(*
SPDX-FileCopyrightText: © 2026 Oleksandr Tiutyk <trofimich@gmail.com>
SPDX-License-Identifier: MIT
License: https://opensource.org/license/mit
*)

(*!
<summary>Formats diagnostics for text-file logging and advances file operations through cyclic execution.</summary>
<description>
Use this backend for buffered text-file output. Direct TryLog and Execute calls on one instance must belong to
one task: its message queue, buffers and file-operation state are not synchronized for concurrent access. For
callers in multiple tasks, use QueuedLogger and let its owner task service this backend; do not bypass the
wrapper with concurrent direct calls. Separate instances writing independently must use separate output files.
Cyclic Execute is required to advance writing and cleanup. Exception logging accepts IReadOnlyException and
reads borrowed diagnostics without transferring ownership. Implementations must not retain exception
references beyond their task cleanup. FAILED is terminal for this instance: no automatic retry or recovery is
provided. Continue calling Execute after failure to discard queued messages, cancel active tasks and release
the send buffer once file operations have finished. Pending messages are not retried. The instance must remain
alive during cleanup. Busy reports pending initialization, messages, file operations or failure cleanup; an
idle open file alone does not make it TRUE. Busy = FALSE does not mean the file handle is closed. After Stop
or in FAILED state, or when the per-instance message queue reaches Parameters.MAX_PENDING_LOG_MESSAGES, all
TryLog methods return FALSE before formatting or queuing new diagnostics. Full-queue rejection preserves
already accepted messages; the current send batch is separate from this limit. Buffered text preserves the
optional message number and category prefix; oversized text is truncated to ERROR_MESSAGE capacity with a
final ellipsis. TryLog methods and Execute do not propagate exceptions. Failed admission returns FALSE;
Execute failures enter FAILED and require further cleanup calls. The terminal allocation latch is preserved
for the task boundary. The initial instance starts automatically through Execute. Stop requests draining of
accepted messages and best-effort file release; continue Execute until STOPPED or until FAILED cleanup
finishes. Start resumes only STOPPED, retaining the file counter and opening the next generated file when a
message arrives. New messages are rejected from Stop until Start. Lifecycle calls belong to the same owner
task as Execute. STOPPED means the close attempt and buffer cleanup finished, not certified physical closure
after a native close error; the underlying resource manager retains its best-effort policy. Embedded task
and resource diagnostics use an owned AdsLogger directly, bypassing LogManager filters/counters and avoiding
feedback into this logger or its QueuedLogger wrapper. maxRecordsPerFile must be positive; zero rejects
admission and the first Execute enters FAILED before any filesystem operation. The configured timeout
applies to directory, open, write and close requests, not to the whole logger lifecycle.
</description>
*)

{attribute 'no_explicit_call' := 'do not call this function block directly'}
FUNCTION_BLOCK SimpleTextFileLogger EXTENDS TOF_Core.Object IMPLEMENTS TOF_Core.ILogger
VAR_STAT
	//! <summary>Static type metadata shared by instances without reading mutable instance state.</summary>
	_ClassName : STRING := __POUNAME();
END_VAR
VAR
	
	{attribute 'hide'} 
	_State : SIMPLE_TEXT_FILE_LOGGER_STATE;
	{attribute 'hide'} 
	_ErrorMessage : TOF_Core.ERROR_MESSAGE;
	{attribute 'hide'}
	_CleanupPending : BOOL;

	//!<summary>
	//! Blocks new messages while accepted work drains and remains set until Start resumes a stopped logger.
	//! </summary>
	_StopRequested : BOOL;
	
	_LogFilePrefix : STRING(32);

	//! <summary>Independent owner-task channel for embedded task and file-resource diagnostics.</summary>
	_InternalDiagnosticLogger : TOF_Core.AdsLogger;

	_CreateDirectoryIfNotExists : TOF_FileSystem.CreateDirectoryIfNotExists(name := "CreateDirectoryIfNotExists");	
	
	_FileContentManager : TOF_FileSystem.FileContentManager(name := "FileContentManager");
	_RecordsPerFile : UINT;
	_WriteBytesTask : TOF_FileSystem.WriteBytesToFile(name := "WriteBytesTask");
	
	_MaxRecordsPerFile : UINT := 100;
	
	_Queue : ARRAY [0..Parameters.MAX_PENDING_LOG_MESSAGES - 1] OF TOF_Core.ERROR_MESSAGE;
	_ReadIndex : UDINT;
	_WriteIndex : UDINT;
	_QueueCount : UDINT;

	_SendBuffer : TOF_Collections.ByteList<0>;
	
	_LogFileCounter : UDINT;
END_VAR

(*!
<summary>Reports the ADS target copied at construction.</summary>
<description>
Directory and file operations use this target; an empty value selects the local system. No I/O is performed.
</description>
*)
{attribute 'monitoring' := 'call'}
PROPERTY AmsNetId : Tc2_System.T_AmsNetID
GET
AmsNetId := _CreateDirectoryIfNotExists.AmsNetId;
END_GET
END_PROPERTY

(*!
<summary>Reports unfinished initialization, message processing, file operations or failure cleanup.</summary>
<description>
TRUE before initialization finishes, while messages or file tasks remain pending, during file acquisition or
release, while a requested normal stop is unfinished, and until failure cleanup completes. An open file
waiting for new messages does not make the logger busy. FALSE does not certify successful writes or a closed
file handle. Continue Execute while cleanup is pending after FAILED.
</description>
*)
{attribute 'monitoring' := 'call'}
PROPERTY Busy : BOOL
GET
Busy := _State = SIMPLE_TEXT_FILE_LOGGER_STATE.INITIAL
	OR_ELSE _State = SIMPLE_TEXT_FILE_LOGGER_STATE.CREATING_DIRECTORY
	OR_ELSE (_StopRequested
		AND_THEN _State <> SIMPLE_TEXT_FILE_LOGGER_STATE.STOPPED
		AND_THEN _State <> SIMPLE_TEXT_FILE_LOGGER_STATE.FAILED)
	OR_ELSE _CleanupPending
	OR_ELSE _QueueCount > TOF_Core.UnsignedInt32.ZERO
	OR_ELSE _FileContentManager.PendingTaskCount > 0
	OR_ELSE _WriteBytesTask.State.Running
	OR_ELSE _WriteBytesTask.FileOperationInProgress
	OR_ELSE (_FileContentManager.State.Running AND_THEN NOT _FileContentManager.RunningSubstate.Processing);
END_GET
END_PROPERTY

(*!
<summary>Provides the concrete logger type name.</summary>
<description>
Returns borrowed read-only initialized static storage. Reading has no side effects or exceptions.
Do not modify the referenced metadata; initialized storage is available before base initialization.
</description>
*)
{attribute 'monitoring' := 'call'}
PROPERTY ClassName : REFERENCE TO STRING
GET
ClassName REF= _ClassName;
END_GET
END_PROPERTY

(*!
<summary>Builds the current log path from the configured directory, prefix, local timestamp and file counter.</summary>
<description>
Uses the existing naming policy without checking for an existing file. A path that exceeds the return capacity
raises StringOverflowException for Execute to report as FAILED. Computes the path on the stack without dynamic
string-builder allocations; no truncated path is used.
</description>
*)
METHOD PRIVATE createCurrentFilePath : Tc2_System.T_MaxString
VAR
	directoryPathText : Tc2_System.T_MaxString;
	timestampText : STRING(32);
	counterText : STRING(16);
	filePathLength : UDINT;
END_VAR
directoryPathText := DirectoryPath;
timestampText := TOF_Core.DateAndTimes.ToString(value := LDT_TO_DT(TOF_Core.System.SystemLocalDateTime));
counterText := TO_STRING(_LogFileCounter);

// Fixed separators and extension '\' + '_' + '_' + '.log' add 7 characters.
filePathLength := TO_UDINT(Tc2_Standard.LEN(STR := directoryPathText))
	+ TO_UDINT(Tc2_Standard.LEN(STR := _LogFilePrefix))
	+ TO_UDINT(Tc2_Standard.LEN(STR := timestampText))
	+ TO_UDINT(Tc2_Standard.LEN(STR := counterText))
	+ 7;

IF filePathLength > 255 THEN
	TOF_Core.Exceptions.ThrowStringOverflow(
		sourceNamespaceName := NamespaceName,
		sourceClassName := ClassName,
		sourcePOUName := __POUNAME(),
		sourcePosition := __POSITION(),
		stringName := 'CurrentFilePath',
		actualLength := filePathLength,
		maxLength := 255
	);  
END_IF

createCurrentFilePath := TOF_Core.Strings.Concat255(
	directoryPathText,
	'\',
	_LogFilePrefix,
	'_',
	timestampText,
	'_',
	counterText,
	'.log');
END_METHOD

(*!
<summary>Reports the copied output directory.</summary>
<description>
The native target resolves this path with DirectoryPathType. Filename generation retains the configured
directory and rejects overflow rather than silently truncating the generated path.
</description>
*)
{attribute 'monitoring' := 'call'}
PROPERTY DirectoryPath : Tc2_System.T_MaxString
GET
DirectoryPath := _CreateDirectoryIfNotExists.DirectoryPath;
END_GET
END_PROPERTY

(*!
<summary>Reports the native path context copied at construction.</summary>
<description>
Used by both directory creation and file opening; this observation does not validate or open a path.
</description>
*)
{attribute 'monitoring' := 'call'}
PROPERTY DirectoryPathType : Tc2_System.E_OpenPath
GET
DirectoryPathType := _CreateDirectoryIfNotExists.PathType;
END_GET
END_PROPERTY

(*!
<summary>Borrows the retained terminal failure diagnostic.</summary>
<description>
Meaningful after State becomes FAILED; cleanup preserves the original diagnostic. The reference remains
valid while this instance lives. Treat it as read-only: ST reference assignment can otherwise mutate it.
Read only from the logger owner task or with external synchronization; no cross-task snapshot is provided.
</description>
*)
{attribute 'monitoring' := 'call'}
PROPERTY ErrorMessage : REFERENCE TO TOF_Core.ERROR_MESSAGE
GET
ErrorMessage REF= _ErrorMessage;
END_GET
END_PROPERTY

(*!
<summary>Advances initialization, writing, requested normal stopping or cleanup after terminal failure.</summary>
<description>
Does not propagate exceptions. On the first failure, enters FAILED and attempts to store the diagnostic. If
diagnostic extraction fails, stores a fixed fallback message without allocating an exception. Subsequent calls
discard queued messages and advance cancellation without starting new writes. The send buffer is released only
after its task and file operation have finished and the manager is no longer running. Cleanup exceptions are
caught; cleanup remains pending for a later call without replacing the original ErrorMessage or recovering the
logger. Fatal allocation state remains latched for the task boundary. After Stop, initialization and already
accepted messages finish normally, including file rotation. Once all writes complete, STOPPING advances
resource release without scheduling further messages. Only then are the manager and write task reset and the
send buffer released before entering STOPPED. A failure during draining uses the existing FAILED path and may
discard unwritten messages. Execute does nothing in STOPPED; Start is required to resume.
</description>
*)
METHOD Execute
VAR	
	exceptionCode : __SYSTEM.ExceptionCode;
	exception : TOF_Core.IException;
END_VAR
VAR
	formattedExceptionMessage : TOF_Core.ERROR_MESSAGE;
END_VAR
__TRY
	stopAfterAllocationFailure();

	IF _State = SIMPLE_TEXT_FILE_LOGGER_STATE.INITIAL
		AND_THEN _MaxRecordsPerFile = TOF_Core.UnsignedInt16.MIN_VALUE
	THEN
		_ErrorMessage := "MaxRecordsPerFile must be greater than zero.";
		_State := SIMPLE_TEXT_FILE_LOGGER_STATE.FAILED;
		_CleanupPending := TRUE;
	END_IF

	IF _State = SIMPLE_TEXT_FILE_LOGGER_STATE.FAILED THEN

		IF NOT _CleanupPending THEN
			RETURN;
		END_IF

		_QueueCount := 0;
		_ReadIndex := 0;
		_WriteIndex := 0;

		IF _CreateDirectoryIfNotExists.State.Running THEN
			_CreateDirectoryIfNotExists.Cancel();
			_CreateDirectoryIfNotExists.Execute();
		END_IF

		IF _FileContentManager.State.Running THEN
			_FileContentManager.Cancel();
			_FileContentManager.Execute();
		END_IF

		IF NOT _CreateDirectoryIfNotExists.State.Running
			AND_THEN NOT _FileContentManager.State.Running
			AND_THEN NOT _WriteBytesTask.State.Running
			AND_THEN NOT _WriteBytesTask.FileOperationInProgress
		THEN
			_FileContentManager.ClearWaitingTasks();

			_WriteBytesTask.SourceBuffer := 0;
			_WriteBytesTask.BytesCountToWrite := 0;
			_SendBuffer.Clear(releaseDynamicMemory := TRUE);
			_CleanupPending := FALSE;
		END_IF

		RETURN;
	END_IF

	CASE _State OF
		SIMPLE_TEXT_FILE_LOGGER_STATE.INITIAL:

			IF _StopRequested AND_THEN _QueueCount = TOF_Core.UnsignedInt32.ZERO THEN
				_State := SIMPLE_TEXT_FILE_LOGGER_STATE.STOPPED;
				RETURN;
			END_IF

			_CreateDirectoryIfNotExists.Reset();

			IF stopAfterAllocationFailure() THEN
				RETURN;
			END_IF

			_CreateDirectoryIfNotExists.Start();

			IF stopAfterAllocationFailure() THEN
				RETURN;
			END_IF

			_State := SIMPLE_TEXT_FILE_LOGGER_STATE.CREATING_DIRECTORY;

		SIMPLE_TEXT_FILE_LOGGER_STATE.CREATING_DIRECTORY:
			_CreateDirectoryIfNotExists.Execute();

			IF stopAfterAllocationFailure() THEN
				RETURN;
			END_IF

			IF _CreateDirectoryIfNotExists.State.Stopped THEN

				IF _CreateDirectoryIfNotExists.FinalStopReason.WorkDone THEN
					_State := SIMPLE_TEXT_FILE_LOGGER_STATE.LOGGING;
				ELSE
					TOF_Core.Exceptions.ThrowStandard(
						sourceNamespaceName := NamespaceName,
						sourceClassName := ClassName,
						sourcePOUName := __POUNAME(),
						sourcePosition := __POSITION(),
						message := "Log directory not created"
					);
				END_IF

			END_IF

		SIMPLE_TEXT_FILE_LOGGER_STATE.LOGGING:
			_FileContentManager.Execute();

			IF stopAfterAllocationFailure() THEN
				RETURN;
			END_IF

			IF _FileContentManager.State.Stopped AND_THEN _FileContentManager.FinalStopReason.Failure THEN
				formattedExceptionMessage := _FileContentManager.FinalStopReason.Message;

				TOF_Core.Exceptions.ThrowStandard(
					sourceNamespaceName := NamespaceName,
					sourceClassName := ClassName,
					sourcePOUName := __POUNAME(),
					sourcePosition := __POSITION(),
					message := formattedExceptionMessage
				);
			END_IF

			processPendingMessages();

			IF stopAfterAllocationFailure() THEN
				RETURN;
			END_IF

			IF _StopRequested
				AND_THEN _QueueCount = TOF_Core.UnsignedInt32.ZERO
				AND_THEN _FileContentManager.PendingTaskCount = TOF_Core.SignedInt32.ZERO
			THEN
				_FileContentManager.StopWhenNoPendingTasks := TRUE;
				_State := SIMPLE_TEXT_FILE_LOGGER_STATE.STOPPING;
			END_IF

		SIMPLE_TEXT_FILE_LOGGER_STATE.STOPPING:
			_FileContentManager.Execute();

			IF stopAfterAllocationFailure() THEN
				RETURN;
			END_IF

			IF _FileContentManager.State.Stopped AND_THEN _FileContentManager.FinalStopReason.Failure THEN
				_ErrorMessage := _FileContentManager.FinalStopReason.Message;
				_State := SIMPLE_TEXT_FILE_LOGGER_STATE.FAILED;
				_CleanupPending := TRUE;
				RETURN;
			END_IF

			IF NOT _FileContentManager.State.Running THEN
				(* No queued write or native I/O remains; borrowed buffer storage may now be released. *)
				_FileContentManager.Reset();

				IF stopAfterAllocationFailure() THEN
					RETURN;
				END_IF

				_FileContentManager.StopWhenNoPendingTasks := FALSE;
				_WriteBytesTask.Reset();

				IF stopAfterAllocationFailure() THEN
					RETURN;
				END_IF

				_WriteBytesTask.SourceBuffer := TOF_Core.Memory.NULL_ADDRESS;
				_WriteBytesTask.BytesCountToWrite := TOF_Core.UnsignedInt32.ZERO;
				_SendBuffer.Clear(releaseDynamicMemory := TRUE);
				_RecordsPerFile := 0;

				_State := SIMPLE_TEXT_FILE_LOGGER_STATE.STOPPED;
			END_IF

	END_CASE

__CATCH(exceptionCode)
	IF _State <> SIMPLE_TEXT_FILE_LOGGER_STATE.FAILED THEN
		_State := SIMPLE_TEXT_FILE_LOGGER_STATE.FAILED;
		_CleanupPending := TRUE;

		__TRY
			exception := TOF_Core.ExceptionManager.GetLastException(
				exceptionCode := exceptionCode,
				catchPointNamespaceName := NamespaceName,
				catchPointPOUName := __POUNAME(),
				catchPointPosition := __POSITION()
			);
			_ErrorMessage := exception.GetMessage();
		__CATCH
			_ErrorMessage := "File logger failed; diagnostic information is unavailable.";
		__ENDTRY

	END_IF

__ENDTRY
END_METHOD

(*!
<summary>Copies logger configuration and binds an independent diagnostic route without performing I/O.</summary>
<description>
All additional constructor arguments must be supplied explicitly. directoryPath and logFilePrefix determine
the existing timestamp/counter filename policy; instances must use separate output files. maxRecordsPerFile
must be positive. Zero is retained without throwing here; TryLog rejects it and Execute reports FAILED before
filesystem I/O. timeout applies to directory, open, write and close requests. Lifecycle initialization only
copies configuration and borrowed routes; it does not create exceptions or invoke diagnostic callbacks.
</description>
<param name="directoryPath">Output directory resolved on the configured ADS target.</param>
<param name="logFilePrefix">Filename prefix copied for this instance.</param>
<param name="maxRecordsPerFile">Positive record count; zero is reported by Execute before I/O.</param>
<param name="directoryPathType">Native path context for directory and file operations.</param>
<param name="timeout">Per-request native timeout for directory, open, write and close.</param>
<param name="amsNetId">ADS target; empty selects the local system.</param>
*)
METHOD FB_init : BOOL
VAR_INPUT
	bInitRetains : BOOL; // TRUE: the retain variables are initialized (reset warm / reset cold)
	bInCopyCode : BOOL;  // TRUE: the instance will be copied to the copy code afterward (online change)
	directoryPath : Tc2_System.T_MaxString;
	logFilePrefix : STRING(32);
	maxRecordsPerFile : UINT;
	directoryPathType : Tc2_System.E_OpenPath; 
	timeout : TIME; 
	amsNetId : Tc2_System.T_AmsNetID; 
END_VAR
_CreateDirectoryIfNotExists.DiagnosticLogger := _InternalDiagnosticLogger;
_FileContentManager.DiagnosticLogger := _InternalDiagnosticLogger;
_WriteBytesTask.DiagnosticLogger := _InternalDiagnosticLogger;
_WriteBytesTask.Timeout := timeout;

_CreateDirectoryIfNotExists.DirectoryPath := directoryPath;
_CreateDirectoryIfNotExists.PathType := directoryPathType;
_CreateDirectoryIfNotExists.Timeout := timeout;
_CreateDirectoryIfNotExists.AmsNetId := amsNetId;

_FileContentManager.PathType := directoryPathType;
_FileContentManager.ModeFlags := Tc2_System.Global_Variables.FOPEN_MODEWRITE
	OR Tc2_System.Global_Variables.FOPEN_MODEPLUS
	OR Tc2_System.Global_Variables.FOPEN_MODETEXT;
_FileContentManager.Timeout := timeout;
_FileContentManager.AmsNetId := amsNetId;

_LogFilePrefix := logFilePrefix;

_MaxRecordsPerFile := maxRecordsPerFile;
END_METHOD

(*!
<summary>Reports the filename prefix copied at construction.</summary>
<description>
Combined with local timestamp and the retained counter; it does not establish exclusive creation or
global uniqueness. Use separate output files for independent logger instances.
</description>
*)
{attribute 'monitoring' := 'call'}
PROPERTY LogFilePrefix : STRING(32)
GET
LogFilePrefix := _LogFilePrefix;
END_GET
END_PROPERTY

(*!
<summary>Reports the positive number of diagnostic records permitted in one generated file.</summary>
<description>
Zero is a configuration error: TryLog rejects admission and Execute records FAILED before filesystem I/O.
The limit counts diagnostic records, not physical lines inside a message; rotation advances on Execute.
</description>
*)
{attribute 'monitoring' := 'call'}
PROPERTY MaxRecordsPerFile : UINT
GET
MaxRecordsPerFile := _MaxRecordsPerFile;
END_GET
END_PROPERTY

(*!
<summary>Borrows the library namespace.</summary>
<description>
Read-only compiler-initialized namespace storage; do not modify the referenced text.
</description>
*)
{attribute 'monitoring' := 'call'}
PROPERTY NamespaceName : REFERENCE TO STRING
GET
NamespaceName REF= CurrentNamespace.Name;
END_GET
END_PROPERTY

(*!
<summary>Transfers queued messages into a batch and schedules its asynchronous file write.</summary>
<description>
Called by Execute. Leaves messages queued while a previous file task or file rotation is pending. Removes
messages from the queue as they are copied into the send buffer, up to the per-file record limit. The send
buffer must remain alive until the write operation finishes. Invalid write-task state and failures from nested
operations propagate to Execute for its failure handling and cleanup. Returning does not mean that the
messages have been written to the file.
</description>
*)
METHOD PRIVATE processPendingMessages
VAR
	formattedExceptionMessage : TOF_Core.ERROR_MESSAGE;
END_VAR
IF _QueueCount = 0 OR_ELSE _FileContentManager.PendingTaskCount > 0 THEN
	RETURN;
END_IF

IF NOT _WriteBytesTask.State.Ready AND_THEN NOT _WriteBytesTask.State.Stopped THEN
	formattedExceptionMessage := TOF_Core.WideStrings.Concat255(
		"WriteBytesTask has invalid state '",
		TO_WSTRING(_WriteBytesTask.State.Value),
		"'"
	);

	TOF_Core.Exceptions.ThrowStandard(
		sourceNamespaceName := NamespaceName,
		sourceClassName := ClassName,
		sourcePOUName := __POUNAME(),
		sourcePosition := __POSITION(),
		message := formattedExceptionMessage
	);
END_IF

IF _WriteBytesTask.State.Stopped AND_THEN NOT _WriteBytesTask.FinalStopReason.WorkDone THEN
	formattedExceptionMessage := TOF_Core.WideStrings.Concat255(
		"WriteBytesTask has invalid stop reason '",
		TO_WSTRING(_WriteBytesTask.FinalStopReason.Value),
		"'"
	);

	TOF_Core.Exceptions.ThrowStandard(
		sourceNamespaceName := NamespaceName,
		sourceClassName := ClassName,
		sourcePOUName := __POUNAME(),
		sourcePosition := __POSITION(),
		message := formattedExceptionMessage
	);
END_IF

IF _RecordsPerFile >= _MaxRecordsPerFile AND_THEN _FileContentManager.State.Running THEN

	IF NOT _FileContentManager.RunningSubstate.ResourceReleasing THEN
		_FileContentManager.Cancel();
	END_IF

	IF _FileContentManager.State.Running THEN
		RETURN;
	END_IF

END_IF

_SendBuffer.Clear();

IF _FileContentManager.FilePath = '' OR_ELSE _RecordsPerFile >= _MaxRecordsPerFile THEN
	_RecordsPerFile := 0;
	_LogFileCounter := _LogFileCounter + 1;

	_FileContentManager.Reset();

	IF stopAfterAllocationFailure() THEN
		RETURN;
	END_IF

	_FileContentManager.FilePath := createCurrentFilePath();

	_FileContentManager.Start();

	IF stopAfterAllocationFailure() THEN
		RETURN;
	END_IF

	_SendBuffer.AppendData(
		data := ADR(TOF_Core.WideStrings.ByteOrderMark),
		dataSize := SIZEOF(TOF_Core.WideStrings.ByteOrderMark)
	);
END_IF

WHILE _QueueCount > 0 DO
	_SendBuffer.AppendData(
		data := ADR(_Queue[_ReadIndex]),
		dataSize := TO_DINT(Tc2_Utilities.WLEN2(pWSTRING := ADR(_Queue[_ReadIndex])) * TOF_Core.WideStrings.CharSize)
	);
	_SendBuffer.AppendData(
		data := ADR(TOF_Core.WideStrings.NewLine),
		dataSize := TO_DINT(SIZEOF(TOF_Core.WideStrings.NewLine) - TOF_Core.WideStrings.CharSize)
	);

	_ReadIndex := _ReadIndex + 1;

	IF _ReadIndex >= Parameters.MAX_PENDING_LOG_MESSAGES THEN
		_ReadIndex := 0;
	END_IF

	_QueueCount := _QueueCount - 1;

	_RecordsPerFile := _RecordsPerFile + 1;

	IF _RecordsPerFile >= _MaxRecordsPerFile THEN
		EXIT;
	END_IF

END_WHILE

_WriteBytesTask.Reset();

IF stopAfterAllocationFailure() THEN
	RETURN;
END_IF

_WriteBytesTask.SourceBuffer := _SendBuffer.DataAddress;
_WriteBytesTask.BytesCountToWrite := TO_UDINT(_SendBuffer.Length);

_FileContentManager.Enqueue(fileHandleTask := _WriteBytesTask);
END_METHOD

(*!
<summary>Reports the size of the concrete logger instance in bytes.</summary>
<description>
Includes the fixed queue and embedded instances; separately allocated dynamic buffers are excluded.
</description>
*)
{attribute 'monitoring' := 'call'}
PROPERTY SelfSize : ULINT
GET
SelfSize := XSIZEOF(THIS^);
END_GET
END_PROPERTY

(*!
<summary>Resumes a normally stopped logger and permits new messages.</summary>
<description>
Call from the owner task. Returns TRUE only from STOPPED; INITIAL already starts automatically, and
initializing, logging, stopping or FAILED instances return FALSE without changing state. Does not perform I/O
or propagate exceptions. Subsequent Execute calls check the directory again. The next accepted message opens
the next generated file using the retained counter, rather than reopening the previous file. This uses the
existing naming policy, not exclusive creation or global name uniqueness. Does not recover a FAILED instance
or certify that an earlier best-effort close succeeded.
</description>
*)
METHOD Start : BOOL
IF _State <> SIMPLE_TEXT_FILE_LOGGER_STATE.STOPPED THEN
	RETURN;
END_IF

_StopRequested := FALSE;
_State := SIMPLE_TEXT_FILE_LOGGER_STATE.INITIAL;
Start := TRUE;
END_METHOD

(*!
<summary>Reports initialization, logging, normal stopping, stopped or terminal failure state.</summary>
<description>
After Stop, the current initialization/logging state persists while accepted messages drain; STOPPING then
denotes final file release. STOPPED permits Start and has no pending writes or buffer cleanup, but does not
certify physical closure after a native close error. FAILED does not recover automatically and rejects new
diagnostics. It does not by itself certify that pending file operations have finished or buffered memory has
been released.
</description>
*)
{attribute 'monitoring' := 'call'}
PROPERTY State : SIMPLE_TEXT_FILE_LOGGER_STATE
GET
State := _State;
END_GET
END_PROPERTY

(*!
<summary>Requests completion of accepted messages followed by normal file release.</summary>
<description>
Call from the owner task. Returns TRUE for an accepted or repeated request, including STOPPED. Returns FALSE
in FAILED, where Execute must instead finish the existing failure cleanup. Immediately rejects new TryLog
calls without discarding accepted messages. Does not perform I/O or propagate exceptions. Continue cyclic
Execute until STOPPED; failures may enter FAILED and discard unwritten messages under its existing cleanup
policy. Start cannot cancel an unfinished stop. Best-effort close completion is not a guarantee of physical
release after a native close error.
</description>
*)
METHOD Stop : BOOL
IF _State = SIMPLE_TEXT_FILE_LOGGER_STATE.FAILED THEN
	RETURN;
END_IF

_StopRequested := TRUE;
Stop := TRUE;
END_METHOD

(*!
<summary>Reports the per-request native timeout copied at construction.</summary>
<description>
Applies to directory enumeration/creation and file open, write and close requests. It is not a deadline
for the whole logger lifecycle or a guarantee of physical release after native failure.
</description>
*)
{attribute 'monitoring' := 'call'}
PROPERTY Timeout : TIME
GET
Timeout := _CreateDirectoryIfNotExists.Timeout;
END_GET
END_PROPERTY

(*!
<summary>Formats an error and queues its text for later file writing.</summary>
<description>
Returns FALSE after Stop or in FAILED state, or when the message queue is full before reading or formatting
the error. An invalid reference is ignored. Otherwise delegates to TryLogMessage; TRUE confirms buffering, not
completion of the file write. Exceptions are caught and reported as FALSE without further logging. The
terminal allocation latch is preserved.
Returns FALSE when fatal allocation state is observed before work or after nested calls. The latch remains
set for the caller's task boundary; already accepted or emitted records are not rolled back.
</description>
<param name="error">Borrowed error to format.</param>
<param name="messageNumber">Optional borrowed number to include in the buffered text.</param>
*)
METHOD TryLogError : BOOL
VAR_INPUT
	error : REFERENCE TO TOF_Core.ERROR;
	messageNumber : REFERENCE TO ULINT := 0;
END_VAR
VAR
	message : TOF_Core.ERROR_MESSAGE;
END_VAR
__TRY

	IF TOF_Core.DynamicMemoryManager.HasAllocationFailed THEN
		RETURN;
	END_IF

	IF _MaxRecordsPerFile = TOF_Core.UnsignedInt16.MIN_VALUE
		OR_ELSE _StopRequested
		OR_ELSE _State = SIMPLE_TEXT_FILE_LOGGER_STATE.FAILED
		OR_ELSE _QueueCount >= Parameters.MAX_PENDING_LOG_MESSAGES
	THEN
		TryLogError := FALSE;
		RETURN;
	END_IF

	IF NOT __ISVALIDREF(error) THEN
		RETURN;
	END_IF

	message := error.ToString(
		sourceDisplayMode := TOF_Core.ERROR_SOURCE_DISPLAY_MODE.HIDDEN,
		timestampDisplayMode := TOF_Core.TIMESTAMP_DISPLAY_MODE.LOCAL
	);

	TryLogError := TryLogMessage(
		category := SEL(
			error.Severity = TOF_Core.ERROR_SEVERITY.CRITICAL,
			TOF_Core.LOG_CATEGORY.ERROR,
			TOF_Core.LOG_CATEGORY.CRITICAL_ERROR
		),
		message := message,
		messageNumber := messageNumber
	);

	IF TOF_Core.DynamicMemoryManager.HasAllocationFailed THEN
		TryLogError := FALSE;
	END_IF

__CATCH
	TryLogError := FALSE;
__ENDTRY
END_METHOD

(*!
<summary>Attempts to log diagnostic information from a read-only exception view.</summary>
<description>
Borrows the exception for the call without clearing it or taking ownership. The exception and its inner causes
must remain live while their diagnostics are read. Logging does not extend their lifetime. Returns FALSE after
Stop or in FAILED state, or when the message queue is full before reading or formatting the exception.
Otherwise TRUE confirms buffering, not completion of the file write. Exceptions are caught and reported as
FALSE without further logging. The terminal allocation latch is preserved.
Returns FALSE when fatal allocation state is observed before work or after nested calls. The latch remains
set for the caller's task boundary; already accepted or emitted records are not rolled back.
</description>
<param name="exception">Exception view to read; null is ignored.</param>
<param name="severity">Severity used to select the log category.</param>
*)
METHOD TryLogException : BOOL
VAR_INPUT
	exception : TOF_Core.IReadOnlyException;
	severity : TOF_Core.ERROR_SEVERITY;
	messageNumber : REFERENCE TO ULINT := 0;
END_VAR
VAR
	message : TOF_Core.ERROR_MESSAGE;
END_VAR
__TRY

	IF TOF_Core.DynamicMemoryManager.HasAllocationFailed THEN
		RETURN;
	END_IF

	IF _MaxRecordsPerFile = TOF_Core.UnsignedInt16.MIN_VALUE
		OR_ELSE _StopRequested
		OR_ELSE _State = SIMPLE_TEXT_FILE_LOGGER_STATE.FAILED
		OR_ELSE _QueueCount >= Parameters.MAX_PENDING_LOG_MESSAGES
	THEN
		TryLogException := FALSE;
		RETURN;
	END_IF

	IF exception = 0 THEN
		RETURN;
	END_IF

	message := exception.GetMessage(showSource := TRUE, timestampDisplayMode := TOF_Core.TIMESTAMP_DISPLAY_MODE.LOCAL);

	TryLogException := TryLogMessage(
		category := SEL(severity = TOF_Core.ERROR_SEVERITY.CRITICAL, TOF_Core.LOG_CATEGORY.ERROR, TOF_Core.LOG_CATEGORY.CRITICAL_ERROR),
		message := message,
		messageNumber := messageNumber
	);

	IF TOF_Core.DynamicMemoryManager.HasAllocationFailed THEN
		TryLogException := FALSE;
	END_IF

__CATCH
	TryLogException := FALSE;
__ENDTRY
END_METHOD

(*!
<summary>Formats a diagnostic and queues its text for later file writing.</summary>
<description>
Returns FALSE after Stop or in FAILED state, or when the queue reaches Parameters.MAX_PENDING_LOG_MESSAGES,
before formatting or allocating buffered text. Queue rejection does not discard previously accepted messages.
Otherwise formats an optional message number followed by the category and message. Preserves the prefixes and
marks truncated text with an ellipsis. Formatting uses local storage without raising a size-overflow
exception. Text admission copies into fixed instance-owned queue storage without heap allocation. Returns TRUE after successful insertion
into the message buffer; this confirms acceptance, not completion of the asynchronous file write. Exceptions
are caught and reported as FALSE without further logging. The terminal allocation latch is preserved.
Returns FALSE when fatal allocation state is observed before work or after nested calls. The latch remains
set for the caller's task boundary; already accepted or emitted records are not rolled back.
</description>
*)
METHOD TryLogMessage : BOOL
VAR_INPUT
	category : TOF_Core.LOG_CATEGORY;	
END_VAR
VAR_IN_OUT CONSTANT
	message : TOF_Core.ERROR_MESSAGE;
END_VAR
VAR_INPUT
	messageNumber : REFERENCE TO ULINT := 0;
END_VAR
VAR
	textToLog : TOF_Core.ERROR_MESSAGE;
END_VAR
__TRY

	IF TOF_Core.DynamicMemoryManager.HasAllocationFailed THEN
		RETURN;
	END_IF

	IF _MaxRecordsPerFile = TOF_Core.UnsignedInt16.MIN_VALUE
		OR_ELSE _StopRequested
		OR_ELSE _State = SIMPLE_TEXT_FILE_LOGGER_STATE.FAILED
		OR_ELSE _QueueCount >= Parameters.MAX_PENDING_LOG_MESSAGES
	THEN
		TryLogMessage := FALSE;
		RETURN;
	END_IF

	IF __ISVALIDREF(messageNumber) THEN
		textToLog := TOF_Core.WideStrings.Concat255(
			TO_WSTRING(TOF_Core.Exceptions.MESSAGE_NUMBER_PREFIX),
			TO_WSTRING(messageNumber),
			TO_WSTRING(TOF_Core.Exceptions.MESSAGE_NUMBER_SUFFIX)
		);
	END_IF

	TOF_Core.WideStrings.Append255(textToLog, "[", TO_WSTRING(category), "] ");
	TOF_Core.WideStrings.AppendFit(targetString := textToLog, sourceString := message);

	_Queue[_WriteIndex] := textToLog;
	_WriteIndex := _WriteIndex + 1;

	IF _WriteIndex >= Parameters.MAX_PENDING_LOG_MESSAGES THEN
		_WriteIndex := 0;
	END_IF

	_QueueCount := _QueueCount + 1;

	TryLogMessage := TRUE;

	IF TOF_Core.DynamicMemoryManager.HasAllocationFailed THEN
		TryLogMessage := FALSE;
	END_IF

__CATCH
	TryLogMessage := FALSE;
__ENDTRY
END_METHOD

(*!
<summary>Records terminal allocation state without raising or replacing an earlier failure.</summary>
<description>
Returns TRUE when the application fatal latch is observed. Marks the logger FAILED and requests cleanup,
preserving an existing failure diagnostic. No allocation or exception creation occurs. Execute must still
advance already pending I/O before releasing its borrowed buffer; the caller supplies the fatal task boundary.
</description>
*)
METHOD PRIVATE stopAfterAllocationFailure : BOOL
IF NOT TOF_Core.DynamicMemoryManager.HasAllocationFailed THEN
	RETURN;
END_IF

IF _State <> SIMPLE_TEXT_FILE_LOGGER_STATE.FAILED THEN
	_ErrorMessage := "File logger stopped after a terminal allocation failure.";
	_State := SIMPLE_TEXT_FILE_LOGGER_STATE.FAILED;
	_CleanupPending := TRUE;
END_IF

stopAfterAllocationFailure := TRUE;
END_METHOD

END_FUNCTION_BLOCK

(* stored: Version 1.1.0.1
   POU SimpleTextFileLogger: Id {83e72a06-d888-49e4-a1fa-5926cd0560d7}, SpecialFunc None
   Folder Service members: Id {31f4dc51-0481-47a0-9f27-e4a804e1bc51}
   Folder Settings: Id {a5c9b4b6-8ecf-4d2a-aad7-cca7912de4af}
   Property AmsNetId: Id {db9518e6-7a39-4ac8-867a-92c65be113ea}
   Get Get: Id {530d554b-478f-4d22-919b-d8853b880ece}
   Property Busy: Id {592a2ef0-f70e-46be-b435-2b32d7b1865a}
   Get Get: Id {369a6e60-cede-41f5-8312-2b57e21b7316}
   Property ClassName: Id {6c5a9607-3c00-4c0a-8401-629f2e4ee076}
   Get Get: Id {0de335d9-e75a-41b2-898b-58ea3af1863b}
   Method createCurrentFilePath: Id {6d3ac00a-486a-4f00-87d7-8b126f05bc66}
   Property DirectoryPath: Id {28aea964-b2f7-4d34-9438-82c3e54285f7}
   Get Get: Id {4d97eb27-ef49-4b43-a312-0269a99b3764}
   Property DirectoryPathType: Id {e71793a7-aadb-4558-8862-be98618eea47}
   Get Get: Id {d6c43e3e-9d0c-4541-99cd-2e8c4518ca4c}
   Property ErrorMessage: Id {5a7d9063-33f0-46e9-a8be-787b9c0b94fb}
   Get Get: Id {8798ddfa-1ff2-4292-a2e0-f047127f13ab}
   Method Execute: Id {17cdfc70-e5ab-42fe-ab86-0d76e3d26166}
   Method FB_init: Id {bc5368c5-4e8b-4212-a2e8-e686311d988e}
   Property LogFilePrefix: Id {146ab0f3-3bee-4300-b03e-e0ac8f4dcd78}
   Get Get: Id {a928530e-14c6-4320-a490-9478edb8bdec}
   Property MaxRecordsPerFile: Id {beb3d3d9-cff4-4690-9465-35ffe8503203}
   Get Get: Id {7fa1b082-aa9d-4ae5-b1bc-a908672be28a}
   Property NamespaceName: Id {4431f0cd-01ee-42e1-822b-47c557994012}
   Get Get: Id {629e0b94-319d-499b-9f3c-7a384bc3cd7b}
   Method processPendingMessages: Id {b3206f74-587e-4877-b310-0e0e64ffdebf}
   Property SelfSize: Id {b9231c56-1285-4e63-ad5b-c9e11184018f}
   Get Get: Id {52d3ef31-002b-4f65-8047-d3dfbc84d9a8}
   Method Start: Id {7a4c4b20-0e3b-4d62-90a5-8d62f5053426}
   Property State: Id {3a575e6f-bb16-4315-8c99-6e30e5beab57}
   Get Get: Id {3db3f673-1f63-4a8b-861c-f15fab2f1187}
   Method Stop: Id {f52fab42-de20-442c-a828-b92d1fc00779}
   Property Timeout: Id {99ab8e8d-9dc9-4652-a5a8-5bf0cbecebc1}
   Get Get: Id {c080a9e4-56eb-4735-8797-b6726b7c34d3}
   Method TryLogError: Id {1ef519f1-badf-441c-b011-cbd27899462a}
   Method TryLogException: Id {e7bb0a19-d38b-4050-ac16-1d13038e54cb}
   Method TryLogMessage: Id {f95238b0-2f26-4019-bd69-7afd783a5817}
   Method stopAfterAllocationFailure: Id {2ce8d69a-5d3b-40c8-bf1b-d96e3d759f40} *)
